// TwinCAT 3 PLC project Dispatch
// ProgramVersion: 3.1.4023.0
// libraries:
//   Tc2_DataExchange, * (Beckhoff Automation GmbH)
//   Tc2_Standard, * (Beckhoff Automation GmbH)
//   Tc2_System, * (Beckhoff Automation GmbH)
//   Tc2_Utilities, * (Beckhoff Automation GmbH)
//   Tc3_BA_Common, * (Beckhoff Automation GmbH)
//   Tc3_Database, * (Beckhoff Automation GmbH)
//   Tc3_Module, * (Beckhoff Automation GmbH)
// project tree:
//   DUTs/ADS/ AdsSocket.TcPOU, FB_Area.TcPOU, Socket.TcDUT, SocketA.TcIO
//   DUTs/Containers/ GenericQueue.TcPOU, IntQueue.TcPOU, PtrQueue.TcPOU, Queue.TcPOU, StringQueue.TcPOU, UnionQ.TcDUT
//   DUTs/Types/ Area.TcDUT, Bundle.TcDUT, Conveyor.TcPOU, Interval.TcDUT, Material.TcDUT (not stored), PositionMaterials.TcDUT
//   DUTs/Enums/ EventsEnum.TcTLEO
//   / GlobalTextList.TcGTLO, PlcTask.TcTTO
//   GVLs/ GVL.TcGVL, Param.TcGVL
//   POUs/ EventLogger.TcPOU, GetBundleRecipe.TcPOU, MAIN.TcPOU
//   POUs/Helper Functions/ AllElementsEqualTo.TcPOU, ArrayContains.TcPOU, ConcatStrings.TcPOU, TimestructToString.TcPOU (not stored)
//   POUs/Obsolete/ Control.TcPOU
// real-time tasks:
//   TASK PlcTask: cycle T#10ms, priority 20, ADS port 350
//   TASK PlcTask1: cycle T#10ms, priority 21, ADS port 351

CONFIGURATION Dispatch
    RESOURCE PLC ON TwinCAT3
        TASK PlcTask(INTERVAL := T#10ms, PRIORITY := 20);
        PROGRAM MAIN WITH PlcTask : MAIN;
    END_RESOURCE
END_CONFIGURATION

// ---- DUTs/ADS/Socket.TcDUT
TYPE Socket :
STRUCT
	localAdr : T_AmsNetId;
	localPort : T_AmsPort;
	
	remoteAdr : T_AmsNetId;
	remotePort : T_AmsPort;
END_STRUCT
END_TYPE

// ---- DUTs/Containers/UnionQ.TcDUT
{attribute 'enable_dynamic_creation'}
TYPE UnionQ :
UNION
	integer : INT;
	float : REAL;
	text : STRING;
	bundle : Bundle;
END_UNION
END_TYPE

(*
this data type is used as the base of GenericQueue
if a data type needs a GenericQueue, add it here
the size of this union is equal to the largest data type in its composition
*)

// ---- DUTs/Types/Area.TcDUT
TYPE Area :
STRUCT
	name : STRING; //area 1, area 2, etc
	id : INT; //name but without area
	
	queue : PtrQueue := (dataSize := SIZEOF(POINTER TO Bundle));
	
	//ready cannot be TRUE if finished is TRUE
	ready : BOOL; //ready to receive
	finished : BOOL; //finished current bundle new bundle
END_STRUCT
END_TYPE

// ---- DUTs/Types/Bundle.TcDUT
{attribute 'enable_dynamic_creation'}
TYPE Bundle :
STRUCT
	id : STRING;
	
	weight : REAL;
	length : USINT;
	width : USINT;
	height : USINT;
	
	pieces : USINT;
	layers : USINT;
	piecesPerLayer : USINT;
	
	extrusionWeight : REAL;
	extrusionHeight : USINT;
	extrusionWidth : USINT;
	
	//processes : (AUTO_RE, AUTO_SS, MAN_RE, MAN_SS);
	reqProcesses : ARRAY[0..3] OF BOOL;
	repack : BOOL;
	currStep : USINT; //for runtime use only
	
	coverPaper : ARRAY[0..1] OF BOOL;
	coverCardboard : ARRAY[0..1] OF BOOL;
	
	paperTop : ARRAY[0..GVL.maxPairs] OF Interval;
	paperLeft : ARRAY[0..GVL.maxPairs] OF Interval;
	paperRight : ARRAY[0..GVL.maxPairs] OF Interval;
	paperBottom : ARRAY[0..GVL.maxPairs] OF Interval;
		
	cardboard : ARRAY[0..GVL.maxPairs] OF PositionMaterials;
	cornerGuard : ARRAY[0..GVL.maxPairs] OF PositionMaterials;
	
	combinedCardboardCornerGuard : ARRAY[0..(GVL.maxPairs*2)] OF PositionMaterials;
	
	chipboard : ARRAY[0..GVL.maxPairs] OF PositionMaterials;
	woodBunk : ARRAY[0..GVL.maxPairs] OF PositionMaterials;
	
	cardboard_over_cornerGuard : BOOL;
	
	//for production log database
	timeStart : TIMESTRUCT;
	timeDone : TIMESTRUCT;
END_STRUCT
END_TYPE

// ---- DUTs/Types/Interval.TcDUT
TYPE Interval :
STRUCT
	startPos : REAL;
	endPos : REAL;
END_STRUCT
END_TYPE

// ---- DUTs/Types/PositionMaterials.TcDUT
TYPE PositionMaterials :
STRUCT
	position : REAL := GVL.nullPos; //default value is set to predefined constant if bundle needs less than 32 position material pairs
	
	top : STRING;
	left : STRING;
	right : STRING;
	bottom : STRING;
	
	topLeft : STRING;
	topLeftFold : USINT;
	
	topRight : STRING;
	topRightFold : USINT;
	
	bottomLeft : STRING;
	bottomLeftFold : USINT;
	
	bottomRight : STRING;
	bottomRightFold : USINT;

	wrapPoints : USINT;
	wrapRotations : USINT;
END_STRUCT
END_TYPE

// ---- DUTs/Enums/EventsEnum.TcTLEO
{attribute 'qualified_only'}
{attribute 'strict'}
{attribute 'to_string'}
TYPE EventsEnum :
(
	//standard operation
	BUNDLE_ADDED_TO_PRODUCTION,
	BUNDLE_RECEIVED,
	BUNDLE_COMPLETE,
	
	//area complete
	AREA_1_COMPLETE,
	AREA_2_COMPLETE,
	AREA_3_COMPLETE,
	AREA_4_COMPLETE,
	AREA_5_COMPLETE,
	AREA_6_COMPLETE,
	
	//area complete
	AREA_1_RECEIVE,
	AREA_2_RECEIVE,
	AREA_3_RECEIVE,
	AREA_4_RECEIVE,
	AREA_5_RECEIVE,
	AREA_6_RECEIVE,

	//standard errors
	BACKLOG,
	MACHINE_FAILURE,
	BUNDLE_EARLY_RECEIVED,
	BUNDLE_LATE_RECEIVED,
	
	AREA_1_DELAY,
	AREA_2_DELAY,
	AREA_3_DELAY,
	AREA_4_DELAY,
	AREA_5_DELAY,
	AREA_6_DELAY,
	
	//robots, motors, database, connections, etc
	CONNECTION_ERROR_PRODUCTION_LOG,
	CONNECTION_ERROR_RECIPE_DB,
	
	CONNECTION_ERROR_AREA_1_DB,
	CONNECTION_ERROR_AREA_2_DB,
	CONNECTION_ERROR_AREA_3_DB,
	CONNECTION_ERROR_AREA_4_DB,
	CONNECTION_ERROR_AREA_5_DB,
	CONNECTION_ERROR_AREA_6_DB,
	
	size
);
END_TYPE

// ---- GVLs/GVL.TcGVL
{attribute 'qualified_only'}
VAR_GLOBAL CONSTANT
	numAreas : USINT := 6;
	
	maxPairs : USINT := 16;
	initArraySize : USINT := 4;
	
	nullPos : REAL := -1;
	
	numMaterials : INT := 32;
	allMaterials : ARRAY[0..numMaterials] OF Material := [
		(code := 'PAP28', width := 28, length := -1),
		
		(code := 'CAR20S', width := 20, length := 30),
		(code := 'CAR20M', width := 20, length := 45),
		(code := 'CAR20L', width := 20, length := 60),
		(code := 'CAR28S', width := 28, length := 30),
		(code := 'CAR28M', width := 28, length := 45),
		(code := 'CAR28L', width := 28, length := 60),
		
		(code := 'COR48', width := 1.5, length := 48),
		(code := 'COR96', width := 1.5, length := 96),
		
		(code := 'CIP18', width := 20, length := 18),
		(code := 'CIP54', width := 20, length := 54),
		
		(code := 'WDT20', width := 20, length := 2.5),
		(code := 'WDT22', width := 22, length := 2.5),
		(code := 'WDT28', width := 28, length := 2.5),
		
		(code := 'WDB20', width := 20, length := 2.5),
		(code := 'WDB22', width := 22, length := 2.5),
		(code := 'WDB28', width := 28, length := 2.5),
		
		(code := 'WDS08', width := 8, length := 2.5),
		(code := 'WDS10', width := 10, length := 2.5),
		(code := 'WDS12', width := 12, length := 2.5),
		(code := 'WDS14', width := 14, length := 2.5),
		(code := 'WDS8x8', width := 16, length := 2.5),
		(code := 'WDS8x10', width := 18, length := 2.5),
		(code := 'WDS20', width := 20, length := 2.5),
		(code := 'WDS22', width := 22, length := 2.5),
		(code := 'WDS12x12', width := 24, length := 2.5),
		(code := 'WDS12x14', width := 26, length := 2.5),
		(code := 'WDS28', width := 28, length := 2.5),
		(code := 'WDS20x10', width := 30, length := 2.5),
		(code := 'WDS20x12', width := 32, length := 2.5),
		
		(code := 'WDW20', width := 20, length := 6),
		(code := 'WDW22', width := 22, length := 6)]; //+1 null material
	
	conveyorLength : REAL;
	precisionTolerance : REAL := 0.05; //in inches
END_VAR
VAR_GLOBAL
	newBundle : Bundle;
	bundleIn AT %I* : Bundle;
	bundleOut AT %Q* : Bundle;
END_VAR

// ---- GVLs/Param.TcGVL
{attribute 'qualified_only'}
VAR_GLOBAL CONSTANT
	initArraySize : UINT := 4;
	
	areaConnections : ARRAY[1..6] OF ARRAY[1..6] OF USINT := [
		[0,0,0,0,5,6],
		[0,0,0,0,0,6],
		[0,0,0,4,5,0],
		[0,0,3,0,5,0],
		[1,0,3,4,0,0],
		[1,2,0,0,0,0]];
		
	
END_VAR

// ---- DUTs/ADS/SocketA.TcIO
INTERFACE SocketA
VAR
	localAdr : T_AmsNetId;
	localPort : T_AmsPort;
END_VAR
VAR
	remoteAdr : T_AmsNetId;
	remotePort : T_AmsPort;
END_VAR

END_INTERFACE

// ---- POUs/MAIN.TcPOU
PROGRAM MAIN
VAR
	newBundle : Bundle; //new bundle, connected to HMI
	
	areas : ARRAY[1..6] OF FB_Area;
	
	bundleIDs : ARRAY[1..6] OF ARRAY[0..16] OF STRING; //for HMI tracking only
	numBundleIDs : ARRAY[1..6] OF ARRAY[0..16] OF UINT; //bundleIDs counter
	
	completedBundles : PtrQueue := (dataSize := SIZEOF(Bundle));
	
	//dbLogger : EventLogger;
	//getBundleFromDB : GetBundleRecipe;
	
	fbSystemTime : FB_LocalSystemTime;
	temp : POINTER TO Bundle; //to push into area queue
END_VAR

//reecive() is called manually by the dispatch operator through the HMI

process(); //track and move bundles between stations

transfer(); //production line output

//HMI parallel processing
//getBundleFromDB(newBundle := newBundle, finished => );

METHOD process : BOOL
VAR
	i : DINT;
	tempBundlePointer : POINTER TO Bundle; //to move data around
	tempBundle : Bundle; //if dereferencing is needed
END_VAR
(*
FOR i:=1 TO 6 BY 1 DO
	IF areas[i].finished THEN
		CASE i OF //add event
			1: dbLogger.addEvent(TO_INT(EventsEnum.AREA_1_COMPLETE));
			2: dbLogger.addEvent(TO_INT(EventsEnum.AREA_2_COMPLETE));
			3: dbLogger.addEvent(TO_INT(EventsEnum.AREA_3_COMPLETE));
			4: dbLogger.addEvent(TO_INT(EventsEnum.AREA_4_COMPLETE));
			5: dbLogger.addEvent(TO_INT(EventsEnum.AREA_5_COMPLETE));
			6: dbLogger.addEvent(TO_INT(EventsEnum.AREA_6_COMPLETE));
		END_CASE
		
		IF i = 1 OR i = 3 OR i = 5 OR i = 6 THEN
			//find next area
			(*
			IF area[next].ready THEN
				temp := areas[i].queue.poll();
				
				//begin transfer, move physical components
				
				area[next].queue.push(temp);
				area[next].ready := FALSE;
				area[next].done := FALSE;
				
				areas[i].done := FALSE;
				areas[i].ready := TRUE;
			END_IF
			*)
		ELSIF i = 2 OR i = 4 THEN //this area is a production endpoint
			tempBundlePointer := areas[i].queue.poll();
			completedBundles.push(tempBundlePointer);
		END_IF
	END_IF
END_FOR
*)
END_METHOD

{attribute 'TcRpcEnable'}
METHOD receive : BOOL
fbSystemTime(
	sNetID := ,
	bEnable := TRUE,
	dwCycle := 5,
	dwOpt := 1,
	tTimeout := DEFAULT_ADS_TIMEOUT,
	bValid => ,
	systemTime => newBundle.timeStart,
	tzId => );

temp := __NEW(Bundle);
MEMCPY(temp, ADR(newBundle), SIZEOF(Bundle));
areas[3].queue.push(temp);

MEMSET(ADR(newBundle), 0, SIZEOF(Bundle)); //clear HMI value

//dbLogger.addEvent(TO_INT(EventsEnum.BUNDLE_ADDED_TO_PRODUCTION));
END_METHOD

METHOD transfer : BOOL
VAR
	i : DINT;
END_VAR
//dbLogger.addEvent(TO_INT(EventsEnum.BUNDLE_ADDED_TO_PRODUCTION));

FOR i:=1 TO GVL.numAreas BY 1 DO
	IF areas[i].done THEN
		areas[i].transfer();
	END_IF
END_FOR
END_METHOD

END_PROGRAM

// ---- DUTs/ADS/FB_Area.TcPOU
FUNCTION_BLOCK FB_Area
VAR
	name : STRING; //fully area name
	id : INT; //area number only
	
	queue : PtrQueue := (dataSize := SIZEOF(POINTER TO Bundle));
	activeBundles : ARRAY[0..10] OF Bundle; //most will only use 1
	capacity : USINT;
	
	ready : BOOL; //ready to receive
	done : BOOL; //finished current bundle new bundle
	
	socket : AdsSocket;
END_VAR
VAR CONSTANT
	test : INT;
END_VAR

METHOD transfer : BOOL
VAR_INPUT
END_VAR
END_METHOD

END_FUNCTION_BLOCK

// ---- DUTs/Containers/Queue.TcPOU
FUNCTION_BLOCK ABSTRACT Queue
VAR
	dataSize : ULINT; //no functionaility, only to force input a type for readability
	varType : __SYSTEM.TYPE_CLASS;
END_VAR
VAR
	elements : FB_BA_DynamicArray := (uiEntrySize := 2, uiMinExpCount := GVL.initArraySize);
	length : USINT := 0;
	uiEntrySizeRef : REFERENCE TO UINT;
END_VAR

END_FUNCTION_BLOCK

// ---- DUTs/Containers/PtrQueue.TcPOU
FUNCTION_BLOCK PtrQueue EXTENDS Queue //stores pointers to bundles, not the bundles themselves
VAR
	//elements : FB_BA_DynamicArray := (uiEntrySize := SIZEOF(PVOID), uiMinExpCount := GVL.initArraySize);
	//length : USINT := 0;
END_VAR

METHOD clear : BOOL
VAR_INPUT
END_VAR
elements.Reset();
length := 0;
END_METHOD

METHOD contains : BOOL
VAR_INPUT
	value : PVOID;
	n : UDINT;
END_VAR
VAR_INST
	i : INT;
END_VAR
IF length = 0 THEN
	contains := FALSE;
	RETURN;
END_IF

FOR i:=0 TO length-1 BY 1 DO
	IF MEMCMP(get(i), value, n) = 0 THEN
		contains := TRUE;
		RETURN;
	END_IF
END_FOR
contains := FALSE;
END_METHOD

METHOD get : PVOID;
VAR_INPUT
	i : UINT;
END_VAR
elements.GetEntry(diIndex := i, pResultEntry := ADR(get));
END_METHOD

METHOD isEmpty : BOOL
VAR_INPUT
END_VAR
isEmpty := (length = 0);
END_METHOD

METHOD poll : PVOID;
VAR_INST
	i : UINT;
END_VAR
poll := get(i := 0);
elements.RemoveEntry(diIndex := 0);
length := length - 1;
END_METHOD

METHOD push : BOOL
VAR_INPUT
	value : PVOID;
END_VAR
elements.AddEntryPtr(pEntry := value);
length := length + 1;
push := TRUE;
END_METHOD

METHOD set : BOOL
VAR_INPUT
	i : INT;
	value : PVOID;
END_VAR
elements.SetEntryPtr(i, value);
END_METHOD

METHOD size : USINT
VAR_INPUT
END_VAR
size := length;
END_METHOD

METHOD sort : BOOL
VAR_INPUT
END_VAR
VAR_INST
	i : INT;
	j : INT;
	temp : INT;
END_VAR
(*FOR i:=0 TO length-1 BY 1 DO
	FOR j:=0 TO length-i-1 BY 1 DO
		IF get(j) > get(j+1) THEN //swap
			temp := get(j);
			set(j, get(j+1));
			set(j+1, temp);
		END_IF
	END_FOR
END_FOR*)
END_METHOD

END_FUNCTION_BLOCK

// ---- DUTs/ADS/AdsSocket.TcPOU
FUNCTION_BLOCK AdsSocket
VAR_STAT
	localPrgName : STRING; //:= GVL.localPrgName;
	localNetId : T_AmsNetId; //:= GVL.localAmsNetId;
	localPort : T_AmsPort; //:= GVL.localAmsPort;
END_VAR
VAR
	remotePrgName : STRING;
	remoteNetId : T_AmsNetId;
	remotePort : T_AmsPort;
END_VAR
VAR
	adsReadSymbol : FB_ReadAdsSymByName;
	adsWriteSymbol : FB_WriteAdsSymByName;
END_VAR

METHOD close : BOOL
remotePrgName := '';
remoteNetId := '';
remotePort := 0;
END_METHOD

METHOD open : BOOL
VAR_INPUT
	newLocalPrgName : STRING;
	newLocalNetId : T_AmsNetId;
	newLocalPort : T_AmsPort;
END_VAR
localPrgName := newLocalPrgName;
localNetId := newLocalNetId;
localPort := newLocalPort;

adsWriteSymbol.sNetId:= remoteNetId;
adsWriteSymbol.nPort:= remotePort;
END_METHOD

METHOD read : BOOL
VAR_INPUT
	symbol : STRING;
	buffer : PVOID;
	symbolSize : UDINT;
END_VAR
adsReadSymbol(
	bRead:= , 
	sNetId:= remoteNetId, 
	nPort:= remotePort, 
	sVarName:= symbol, 
	nDestAddr:= buffer, 
	nLen:= symbolSize, 
	tTimeout:= , 
	eComMode:= , 
	bClearOnError:= TRUE, 
	bBusy=> , 
	bError=> , 
	nErrorId=> );
	
adsReadSymbol.bRead := FALSE;
END_METHOD

METHOD ready : BOOL
ready := (
	remotePrgName <> '' AND
	remoteNetId <> '' AND
	remotePort <> 0);
END_METHOD

METHOD setup : BOOL
localPrgName := '';
localNetId := '';
localPort := 0;

//fill these values with data
END_METHOD

METHOD write : BOOL
VAR_INPUT
	symbol : STRING;
	data : PVOID;
	dataSize : UDINT;
END_VAR
adsWriteSymbol(
	bWrite:= TRUE, 
	sNetId:= remoteNetId, 
	nPort:= remotePort, 
	sVarName:= symbol, 
	nSrcAddr:= data, 
	nLen:= dataSize, 
	tTimeout:= , 
	eComMode:= , 
	bBusy=> , 
	bError=> , 
	nErrorId=> );
	
adsWriteSymbol.bWrite := FALSE;
END_METHOD

END_FUNCTION_BLOCK

// ---- DUTs/Containers/GenericQueue.TcPOU
FUNCTION_BLOCK GenericQueue
VAR_INPUT CONSTANT
	dataSize : UDINT; //no functionaility, only to force input a type for readability
END_VAR
VAR //pointers = 8 byte integers
	elements : FB_BA_DynamicArray := (uiEntrySize := SIZEOF(POINTER TO UnionQ), uiMinExpCount := GVL.initArraySize);
	length : USINT := 0;
END_VAR

METHOD clear : BOOL
VAR_INPUT
END_VAR
elements.Reset();
length := 0;
END_METHOD

METHOD contains : BOOL
VAR_INPUT
	value : UnionQ;
END_VAR
VAR_INST
	i : INT;
END_VAR
IF length = 0 THEN
	contains := FALSE;
	RETURN;
END_IF

FOR i:=0 TO length-1 BY 1 DO
	IF MEMCMP(get(i), ADR(value), SIZEOF(UnionQ)) = 0 THEN
		contains := TRUE;
		RETURN;
	END_IF
END_FOR
contains := FALSE;
END_METHOD

METHOD get : POINTER TO UnionQ
VAR_INPUT
	i : INT;
END_VAR
IF length = 0 OR i < 0 OR i >= length THEN
	get := 0;
ELSE
	elements.GetEntry(diIndex := i, pResultEntry := ADR(get));
END_IF
END_METHOD

METHOD isEmpty : BOOL
VAR_INPUT
END_VAR
isEmpty := length = 0;
END_METHOD

METHOD poll : POINTER TO UnionQ
VAR
	temp : POINTER TO UnionQ;
	i : INT;
END_VAR
poll := get(i := 0);

IF length > 0 THEN
	elements.RemoveEntry(diIndex := 0);
	length := length - 1;
END_IF
END_METHOD

METHOD push : BOOL
VAR_INPUT
	value : POINTER TO UnionQ;
END_VAR
elements.AddEntry(pEntry := ADR(value));
length := length + 1;
END_METHOD

METHOD set : BOOL
VAR_INPUT
	i : INT;
	value : POINTER TO UnionQ;
END_VAR
IF i > 0 AND i < length THEN
	elements.SetEntry(i, ADR(value));
	set := TRUE;
END_IF
END_METHOD

METHOD size : USINT
size := length;
END_METHOD

END_FUNCTION_BLOCK

// ---- DUTs/Containers/IntQueue.TcPOU
FUNCTION_BLOCK IntQueue EXTENDS Queue
VAR
	//elements : FB_BA_DynamicArray := (uiEntrySize :=1, uiMinExpCount := GVL.initArraySize);
END_VAR

uiEntrySizeRef REF= elements.uiEntrySize;
uiEntrySizeRef := TO_UINT(dataSize);

METHOD clear : BOOL
VAR_INPUT
END_VAR
elements.Reset();
length := 0;
END_METHOD

METHOD contains : BOOL
VAR_INPUT
	value : INT;
END_VAR
VAR_INST
	i : INT;
END_VAR
IF length = 0 THEN
	contains := FALSE;
	RETURN;
END_IF

FOR i:=0 TO length-1 BY 1 DO
	IF get(i) = value THEN
		contains := TRUE;
		RETURN;
	END_IF
END_FOR
contains := FALSE;
END_METHOD

METHOD get : INT
VAR_INPUT
	i : INT;
END_VAR
elements.GetEntry(diIndex := i, pResultEntry := ADR(get));
END_METHOD

METHOD isEmpty : BOOL
VAR_INPUT
END_VAR
isEmpty := (length = 0);
END_METHOD

METHOD poll : INT
VAR_INST
	temp : INT;
	i : INT;
END_VAR
temp := get(i := 0);
elements.RemoveEntry(diIndex := 0);
length := length - 1;
poll := temp;
END_METHOD

METHOD push : BOOL
VAR_INPUT
	value : INT;
END_VAR
elements.AddEntry(pEntry := ADR(value));
length := length + 1;
END_METHOD

METHOD set : BOOL
VAR_INPUT
	i : INT;
	value : INT;
END_VAR
elements.SetEntry(i, ADR(value));
END_METHOD

METHOD size : USINT
VAR_INPUT
END_VAR
size := length;
END_METHOD

METHOD sort : BOOL
VAR_INPUT
END_VAR
VAR_INST
	i : INT;
	j : INT;
	temp : INT;
END_VAR
FOR i:=0 TO GVL.maxPairs BY 1 DO
	FOR j:=0 TO GVL.maxPairs BY 1 DO
		IF get(j) > get(j+1) THEN //swap
			temp := get(j);
			set(j, get(j+1));
			set(j+1, temp);
		END_IF
	END_FOR
END_FOR
END_METHOD

END_FUNCTION_BLOCK

// ---- DUTs/Containers/StringQueue.TcPOU
FUNCTION_BLOCK StringQueue EXTENDS Queue
VAR
	elements : FB_BA_DynamicArray := (uiEntrySize := SIZEOF(STRING), uiMinExpCount := GVL.initArraySize);
	//length : USINT := 0;
END_VAR

METHOD get : STRING
VAR_INPUT
	i : UINT;
END_VAR
elements.GetEntry(diIndex := i, pResultEntry := ADR(get));
END_METHOD

METHOD isEmpty : BOOL
VAR_INPUT
END_VAR
isEmpty := (length = 0);
END_METHOD

METHOD poll : STRING
VAR_INST
	temp : STRING;
	i : UINT;
END_VAR
temp := get(i := 0);
elements.RemoveEntry(diIndex := 0);
length := length - 1;
poll := temp;
END_METHOD

METHOD push : BOOL
VAR_INPUT
	value : STRING;
END_VAR
elements.AddEntry(pEntry := ADR(value));
length := length + 1;
END_METHOD

METHOD size : USINT
VAR_INPUT
END_VAR
size := length;
END_METHOD

END_FUNCTION_BLOCK

// ---- DUTs/Types/Conveyor.TcPOU
FUNCTION_BLOCK Conveyor
VAR
	position : REAL;
	velocity : REAL;
	
	retracted : BOOL; //vertical conveyors
END_VAR

METHOD backward : BOOL
VAR_INPUT
END_VAR
END_METHOD

METHOD extend : BOOL
VAR_INPUT
END_VAR
END_METHOD

METHOD forward : BOOL
VAR_INPUT
END_VAR
END_METHOD

METHOD getPosition : REAL;
VAR_INPUT
END_VAR
getPosition := position;
END_METHOD

METHOD getVelocity : REAL;
VAR_INPUT
END_VAR
getVelocity := velocity;
END_METHOD

METHOD reset : BOOL
VAR_INPUT
END_VAR
position := 0;
velocity := velocity; //no change

extend();
END_METHOD

METHOD retract : BOOL
VAR_INPUT
END_VAR
END_METHOD

METHOD target : BOOL
VAR_INPUT
	targetPosition : REAL;
END_VAR
END_METHOD

END_FUNCTION_BLOCK

// ---- POUs/EventLogger.TcPOU
FUNCTION_BLOCK EventLogger//database logging, to be replaced with inbuilt eventlogger
VAR_INPUT
	
END_VAR
VAR
	//client : REFERENCE TO AdsUnit; //some other protocol
	
	completedBundles : REFERENCE TO PtrQueue;
	
	events : IntQueue := (dataSize := 4, varType := __SYSTEM.TYPE_CLASS.TYPE_STRING); //local events queue
	
	fbSQLCommand : FB_SQLCommandEvt(sNetID := '', tTimeout := T#5S);
	fbSQLDatabase : FB_SQLDatabaseEvt (sNetID := '', tTimeout := T#5S);
	fbSQLResult: FB_SQLResultEvt(sNetID:='', tTimeout:=T#5S);
	
	queryOpening : STRING(500) := 'INSERT INTO EventLog(Timestamp, Machine, Event, Type) VALUES(';
	fullQuery : STRING(500);
	
	//for timestamps
	ntSystemTime : NT_GetTime;
    timeAsStruct : TIMESTRUCT;
	
	exeIn : ARRAY [0..2] OF STRING(255);
	
	//iterators
	i : SINT := 0;
	
	//step switch
	step : (IDLE,
			CONNECT_TO_DB, CREATE_CMD, INSERT_CMD, CLOSE_CONNECTION, 
			CONNECT_TO_LOCAL_DB, CREATE_LOCAL_CMD, INSERT_LOCAL_CMD, CLOSE_LOCAL_CONNECTION,
			ERROR);
END_VAR

CASE step OF //1-4 for local DB, 11-14 for plant DB
	//local EventLog DB should store all events for diagnosis
	IDLE:
		IF NOT events.isEmpty() THEN
			step := CONNECT_TO_DB;
		END_IF
		
	CONNECT_TO_DB: //open connection to local EventLog DB
		IF connectToDb() THEN
			step := 1;
		END_IF
		
	CREATE_CMD: //create command
		IF createCommand() THEN
			step := 2;
		END_IF
		
	INSERT_CMD: //insert command
		//timestamp, event, machine, type
		//ntSystemTime(NETID := , START := TRUE, TMOUT := DEFAULT_ADS_TIMEOUT, BUSY => , ERR =>, ERRID =>, TIMESTR => timeAsStruct);
		
		fullQuery := CONCAT(queryOpening, '$''); //timestamp
		fullQuery := CONCAT(fullQuery, TimestructToString(GVL.bundleOut.timeDone));
		fullQuery := CONCAT(fullQuery, '$', ');
		
		exeIn[0] := CONCAT(queryOpening, '$''); //timestamp
		exeIn[0] := CONCAT(fullQuery, TimestructToString(timeAsStruct));
		exeIn[0] := CONCAT(fullQuery, '$', ');
		
		CASE events.get(i:=0) OF //event
			(*EventsEnum.BUNDLE_SENT:
				exeIn[1] := CONCAT(exeIn[1], '$'Bundle Sent (');
				exeIn[1] := CONCAT(exeIn[1], GVL.bundleOut^.id);
				exeIn[1] := CONCAT(exeIn[1], ')$'');*)
			EventsEnum.BACKLOG:
				exeIn[1] := CONCAT(exeIn[1], '$'Backlog$'');
			EventsEnum.MACHINE_FAILURE: //and other specific events to be logged
				exeIn[1] := CONCAT(exeIn[1], '$'Machine Failure$'');
			(*
			EventsEnum.DELAY:
				exeIn[1] := CONCAT(exeIn[1], '$'Delay (');
				exeIn[1] := CONCAT(exeIn[1], GVL.bundleOut.id);
				exeIn[1] := CONCAT(exeIn[1], ')$'');
			*)
			EventsEnum.BUNDLE_LATE_RECEIVED:
				exeIn[1] := CONCAT(exeIn[1], '$'Late Arrival (');
				exeIn[1] := CONCAT(exeIn[1], GVL.bundleOut.id);
				exeIn[1] := CONCAT(exeIn[1], ')$'');
			EventsEnum.BUNDLE_EARLY_RECEIVED:
				exeIn[1] := CONCAT(exeIn[1], '$'Early Arrival (');
				exeIn[1] := CONCAT(exeIn[1], GVL.bundleOut.id);
				exeIn[1] := CONCAT(exeIn[1], ')$'');
			ELSE
				exeIn[1] := CONCAT(exeIn[1], '$'Other/Unknown$'');
		END_CASE
		
		exeIn[2] := CONCAT(exeIn[2], '$'Area 2$')'); //machine
		
		//ADSLOGSTR(msgCtrlMask := ADSLOG_MSGTYPE_ERROR OR ADSLOG_MSGTYPE_MSGBOX, msgFmtStr := sCMD, strArg := strSFCErrorStep);
		
		FOR i:=0 TO 2 BY 1 DO
			fullQuery := CONCAT(fullQuery, exeIn[i]);
		END_FOR
		
		IF fbSQLCommand.Execute(ADR(fullQuery), SIZEOF(fullQuery)) THEN
			step := 3;
		END_IF
	
	//3: //send data to system EventLog DB via TCP client
		(*IF client.send(sAction := 'log event', sData := sCMD) THEN
			step := 4;
		END_IF*)
		
	CLOSE_CONNECTION: //close connection
		events.poll();
		IF fbSQLDatabase.Disconnect() THEN
			step := 100;
		END_IF
	
	//system EventLog DB should only store simplified events
	(*100:
		IF NOT events.isEmpty() THEN
			IF fbSQLDatabase.Connect(5) THEN
				step := 11;
			END_IF
		END_IF
	
	101:
		IF fbSQLDatabase.CreateCmd(ADR(fbSQLCommand)) THEN
			step := 12;
		END_IF
	
	102:
		sCMD := CONCAT(CMD_0, '$''); //timestamp
		sCMD := CONCAT(sCMD, helper.timestructToString(timeAsStruct));
		sCMD := CONCAT(sCMD, '$', ');
		
		CASE events.get(i := 0) OF //event
			EventsEnum.BUNDLE_SENT:
				sCMD := CONCAT(sCMD, '$'Bundle Sent (');
				sCMD := CONCAT(sCMD, GVL.bundleOut^.id);
				sCMD := CONCAT(sCMD, ')$'');
			EventsEnum.BACKLOG:
				sCMD := CONCAT(sCMD, '$'Backlog$'');
			EventsEnum.MACHINE_FAILURE:
				sCMD := CONCAT(sCMD, '$'Machine Failure$'');
			EventsEnum.DELAY:
				sCMD := CONCAT(sCMD, '$'Delay (');
				sCMD := CONCAT(sCMD, GVL.bundleOut^.id);
				sCMD := CONCAT(sCMD, ')$'');
			EventsEnum.BUNDLE_LATE_RECEIVED:
				sCMD := CONCAT(sCMD, '$'Late Arrival (');
				sCMD := CONCAT(sCMD, GVL.bundleOut^.id);
				sCMD := CONCAT(sCMD, ')$'');
			EventsEnum.BUNDLE_EARLY_RECEIVED:
				sCMD := CONCAT(sCMD, '$'Early Arrival (');
				sCMD := CONCAT(sCMD, GVL.bundleOut^.id);
				sCMD := CONCAT(sCMD, ')$'');
			ELSE
				sCMD := CONCAT(sCMD, '$'Other/Unknown$'');
		END_CASE
		
		sCMD := CONCAT(sCMD, '$'Area 2$')'); //machine
		
		ADSLOGSTR(msgCtrlMask := ADSLOG_MSGTYPE_ERROR OR ADSLOG_MSGTYPE_MSGBOX, msgFmtStr := sCMD, strArg := strSFCErrorStep);
		
		IF fbSQLCommand.Execute(ADR(sCMD), SIZEOF(sCMD)) THEN
			step := 3;
		END_IF
	
	103:
		
	104:*)
		
		
END_CASE

METHOD addEvent : BOOL
VAR_INPUT
	event : INT;
END_VAR
events.push(event);
END_METHOD

METHOD connectToDb : BOOL
VAR_INPUT
END_VAR
IF fbSQLDatabase.Connect(1) THEN
	connectToDb := TRUE;
	RETURN;
END_IF
END_METHOD

METHOD createCommand : BOOL
VAR_INPUT
END_VAR
IF fbSQLDatabase.CreateCmd(ADR(fbSQLCommand)) THEN
	createCommand := TRUE;
	RETURN;
END_IF
END_METHOD

METHOD insertCommand : BOOL
VAR_INPUT
END_VAR
VAR_INST
	tempPtr : POINTER TO Bundle;
END_VAR
//for bundle completion events use bundle.timeDone, otherwise use system time
IF events.get(i:=0) = EventsEnum.BUNDLE_COMPLETE THEN
	tempPtr := completedBundles.poll();
	timeAsStruct := tempPtr^.timeDone;
	__DELETE(tempPtr);
ELSE
	ntSystemTime(NETID := , START := TRUE, TMOUT := DEFAULT_ADS_TIMEOUT, BUSY => , ERR =>, ERRID =>, TIMESTR => timeAsStruct);
END_IF

fullQuery := CONCAT(queryOpening, '$''); //timestamp
fullQuery := CONCAT(fullQuery, TimestructToString(GVL.bundleOut.timeDone));
fullQuery := CONCAT(fullQuery, '$', ');

exeIn[0] := CONCAT(queryOpening, '$''); //timestamp
exeIn[0] := CONCAT(fullQuery, TimestructToString(timeAsStruct));
exeIn[0] := CONCAT(fullQuery, '$', ');

CASE events.get(i:=0) OF //event
	(*EventsEnum.BUNDLE_SENT:
		exeIn[1] := CONCAT(exeIn[1], '$'Bundle Sent (');
		exeIn[1] := CONCAT(exeIn[1], GVL.bundleOut^.id);
		exeIn[1] := CONCAT(exeIn[1], ')$'');*)
	EventsEnum.BACKLOG:
		exeIn[1] := CONCAT(exeIn[1], '$'Backlog$'');
	EventsEnum.MACHINE_FAILURE: //and other specific events to be logged
		exeIn[1] := CONCAT(exeIn[1], '$'Machine Failure$'');
	(*
	EventsEnum.DELAY:
		exeIn[1] := CONCAT(exeIn[1], '$'Delay (');
		exeIn[1] := CONCAT(exeIn[1], GVL.bundleOut.id);
		exeIn[1] := CONCAT(exeIn[1], ')$'');
	*)
	EventsEnum.BUNDLE_LATE_RECEIVED:
		exeIn[1] := CONCAT(exeIn[1], '$'Late Arrival (');
		exeIn[1] := CONCAT(exeIn[1], GVL.bundleOut.id);
		exeIn[1] := CONCAT(exeIn[1], ')$'');
	EventsEnum.BUNDLE_EARLY_RECEIVED:
		exeIn[1] := CONCAT(exeIn[1], '$'Early Arrival (');
		exeIn[1] := CONCAT(exeIn[1], GVL.bundleOut.id);
		exeIn[1] := CONCAT(exeIn[1], ')$'');
	ELSE
		exeIn[1] := CONCAT(exeIn[1], '$'Other/Unknown$'');
END_CASE

exeIn[2] := CONCAT(exeIn[2], '$'Area 2$')'); //machine

//ADSLOGSTR(msgCtrlMask := ADSLOG_MSGTYPE_ERROR OR ADSLOG_MSGTYPE_MSGBOX, msgFmtStr := sCMD, strArg := strSFCErrorStep);
END_METHOD

END_FUNCTION_BLOCK

// ---- POUs/GetBundleRecipe.TcPOU
FUNCTION_BLOCK GetBundleRecipe //get bundle data using ID from HMI
VAR_INPUT
	newBundle : REFERENCE TO Bundle;
END_VAR
VAR
	cmd : ARRAY[0..18] OF STRING(5000);
	query : STRING(5000);
	
	fbSQLCommand : FB_SQLCommandEvt(sNetID := '', tTimeout := T#5S);
	fbSQLDatabase : FB_SQLDatabaseEvt(sNetID := '', tTimeout := T#5S);
	fbSQLResult: FB_SQLResultEvt(sNetID := '', tTimeout := T#5S);
	
	dbCheckStep : (CONNECT, READY, EXECUTE, FINISH);
END_VAR
VAR_OUTPUT
	finished : BOOL;
END_VAR

CASE dbCheckStep OF
	CONNECT:
		IF fbSQLDatabase.Connect(1) THEN
			IF NOT fbSqlDatabase.bError THEN
				dbCheckStep := READY;
			END_IF
		END_IF
		
	READY:
		IF fbSQLDatabase.CreateCmd(ADR(fbSQLCommand)) THEN
			dbCheckStep := EXECUTE;
		END_IF
	
	EXECUTE:
		cmd[0] := 'SELECT ';
		cmd[1] := 'weight, length, width, height, pieces, layers, piecesPerLayer, extrusionWeight, extrusionHeight, extrusionWidth, processes'; 
		cmd[2] := 'FROM "Bundle Data - Prototype" WHERE BundleID = $'';
		cmd[3] := TO_STRING(GVL.newBundle.id);
		cmd[4] := '$'';
		query := ConcatStrings(cmd, '', '', '');
		
		IF fbSQLCommand.ExecuteDataReturn(ADR(query), SIZEOF(query), ADR(fbSqlResult)) THEN
			dbCheckStep := FINISH;
		END_IF
		
	FINISH:
		fbSqlResult.Read(0, 1, ADR(newBundle), SIZEOF(Bundle), TRUE, FALSE);
			
		IF fbSQLDatabase.Disconnect() THEN
			fbSqlResult.Release();
			finished := TRUE;
			dbCheckStep := CONNECT;
		END_IF
END_CASE

END_FUNCTION_BLOCK

// ---- POUs/Helper Functions/ConcatStrings.TcPOU
FUNCTION ConcatStrings : STRING(5000)
VAR_IN_OUT
	stringsArr : ARRAY[*] OF STRING(5000);
END_VAR
VAR_INPUT
	opening : STRING(5000);
	closing : STRING(5000);
	separator : STRING(5000);
END_VAR
VAR
	fullString : STRING(5000);
	i : DINT := 0;	
END_VAR

fullString := opening; //opening segment

FOR i:=LOWER_BOUND(stringsArr, 1) TO UPPER_BOUND(stringsArr, 1)-1 BY 1 DO //first element to 2nd last element
	CONCAT2(ADR(fullString), ADR(stringsArr[i]), ADR(fullString), SIZEOF(fullString));
	CONCAT2(ADR(fullString), ADR(separator), ADR(fullString), SIZEOF(fullString));
END_FOR
CONCAT2(ADR(fullString), ADR(stringsArr[UPPER_BOUND(stringsArr, 1)]), ADR(fullString), SIZEOF(fullString)); //final element

CONCAT2(ADR(fullString), ADR(closing), ADR(fullString), SIZEOF(fullString)); //closing segment

concatStrings := fullString;

END_FUNCTION

// ---- POUs/Helper Functions/AllElementsEqualTo.TcPOU
FUNCTION AllElementsEqualTo : BOOL
VAR_IN_OUT
	arr : ARRAY[*] OF INT;
END_VAR
VAR_INPUT
	firstIndex : SINT;
	lastIndex : SINT;
	value : INT;
END_VAR
VAR
	i : SINT := 0;
END_VAR

FOR i:=firstIndex TO lastIndex BY 1 DO
	IF NOT arr[i] = value THEN
		allElementsEqualTo := FALSE;
		RETURN;
	END_IF
END_FOR

allElementsEqualTo := TRUE;
RETURN;

END_FUNCTION

// ---- POUs/Helper Functions/ArrayContains.TcPOU
FUNCTION ArrayContains : BOOL
VAR_IN_OUT
	arr : ARRAY[*] OF INT;
END_VAR
VAR_INPUT
	firstIndex : SINT;
	lastIndex : SINT;
	value : INT;
END_VAR
VAR
	i : SINT := 0;
END_VAR

FOR i:=firstIndex TO lastIndex BY 1 DO
	IF arr[i] = value THEN
		arrayContains := TRUE;
		RETURN;
	END_IF
END_FOR

arrayContains := FALSE;

END_FUNCTION

// ---- POUs/Obsolete/Control.TcPOU
FUNCTION_BLOCK Control
VAR
	newBundle : Bundle; //new bundle, connected to HMI
	
	areas : ARRAY[1..6] OF Area;
	
	bundleIDs : ARRAY[1..6] OF ARRAY[0..16] OF STRING; //for HMI tracking only
	numBundleIDs : ARRAY[1..6] OF ARRAY[0..16] OF UINT; //bundleIDs counter
	
	completedBundles : PtrQueue := (dataSize := SIZEOF(Bundle));
	
	
	//dbLogger : EventLogger;
	//getBundleFromDB : GetBundleRecipe;
	
	fbSystemTime : FB_LocalSystemTime;
	temp : POINTER TO Bundle; //to push into area queue
END_VAR

//reecive() is called manually by the dispatch operator through the HMI

process(); //track and move bundles between stations

transfer(); //production line output

//HMI parallel processing
//getBundleFromDB(newBundle := newBundle, finished => );

METHOD process : BOOL
VAR_INST
	i : DINT;
	tempBundlePointer : POINTER TO Bundle; //to move data around
	tempBundle : Bundle; //if dereferencing is needed
END_VAR
(*
FOR i:=1 TO 6 BY 1 DO
	IF areas[i].finished THEN
		CASE i OF //add event
			1: dbLogger.addEvent(TO_INT(EventsEnum.AREA_1_COMPLETE));
			2: dbLogger.addEvent(TO_INT(EventsEnum.AREA_2_COMPLETE));
			3: dbLogger.addEvent(TO_INT(EventsEnum.AREA_3_COMPLETE));
			4: dbLogger.addEvent(TO_INT(EventsEnum.AREA_4_COMPLETE));
			5: dbLogger.addEvent(TO_INT(EventsEnum.AREA_5_COMPLETE));
			6: dbLogger.addEvent(TO_INT(EventsEnum.AREA_6_COMPLETE));
		END_CASE
		
		IF i = 1 OR i = 3 OR i = 5 OR i = 6 THEN
			//find next area
			(*
			IF area[next].ready THEN
				temp := areas[i].queue.poll();
				
				//begin transfer, move physical components
				
				area[next].queue.push(temp);
				area[next].ready := FALSE;
				area[next].done := FALSE;
				
				areas[i].done := FALSE;
				areas[i].ready := TRUE;
			END_IF
			*)
		ELSIF i = 2 OR i = 4 THEN //this area is a production endpoint
			tempBundlePointer := areas[i].queue.poll();
			completedBundles.push(tempBundlePointer);
		END_IF
	END_IF
END_FOR
*)
END_METHOD

{attribute 'TcRpcEnable'}
METHOD receive : BOOL
fbSystemTime(
	sNetID := ,
	bEnable := TRUE,
	dwCycle := 5,
	dwOpt := 1,
	tTimeout := DEFAULT_ADS_TIMEOUT,
	bValid => ,
	systemTime => newBundle.timeStart,
	tzId => );

temp := __NEW(Bundle);
MEMCPY(temp, ADR(newBundle), SIZEOF(Bundle));
areas[3].queue.push(temp);

MEMSET(ADR(newBundle), 0, SIZEOF(Bundle)); //clear HMI value

//dbLogger.addEvent(TO_INT(EventsEnum.BUNDLE_ADDED_TO_PRODUCTION));
END_METHOD

METHOD transfer : BOOL
//dbLogger.addEvent(TO_INT(EventsEnum.BUNDLE_ADDED_TO_PRODUCTION));
END_METHOD

END_FUNCTION_BLOCK
